FUNCTION TaskHeartbeat : BOOL;
VAR_INPUT
	update		: BOOL;
END_VAR
VAR_STAT
	_beat		: BOOL;
END_VAR


IF (update) THEN
	_beat := NOT _beat;
END_IF

TaskHeartbeat := _beat;

END_FUNCTION

(* stored: Version 1.1.0.1, ProductVersion 3.1.4024.12
   POU TaskHeartbeat: Id {d973c915-447b-480e-a34b-22f0c4d74dca}, SpecialFunc None *)
